// TIA Portal V17 export
// export: Created 2023-04-04T07:17:24.6561318Z, ExportSetting WithDefaults, DisplayName Totally Integrated Automation Portal, DisplayVersion V17 Update 4, DisplayName TIA Portal Openness, DisplayVersion V17 Update 4, DisplayName TIA Portal Version Control Interface, DisplayVersion V17, DisplayName STEP 7 Professional, DisplayVersion V17 Update 4, DisplayName STEP 7 Safety, DisplayVersion V17, DisplayName WinCC Professional, DisplayVersion V17 Update 4
FUNCTION "NTP" : Void   // FC124, LAD
{ S7_Optimized_Access := 'TRUE' }
VERSION : 0.1
// stored: AutoNumber false, IsIECCheckEnabled false, SetENOAutomatically false, UDAEnableTagReadback false
   VAR_TEMP   // added for the SCL form of the ladder/FBD networks
      _w1 : Bool;
   END_VAR
BEGIN

REGION Network 1: Server NTP
   // To run also in a task 1s, it's used by the MINI_PC to retrieve the correct date and time
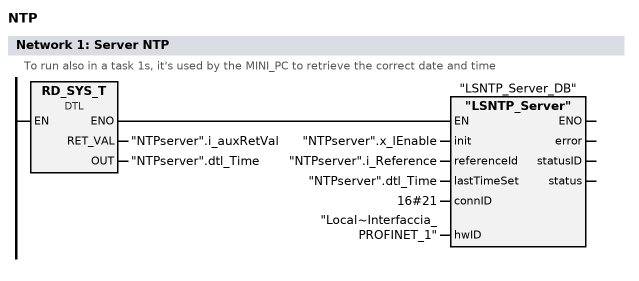
   RUNG wire#powerrail
      { S7_Templates := "date_type := DTL" } RD_SYS_T(RET_VAL => "NTPserver".i_auxRetVal, OUT => "NTPserver".dtl_Time)
      "LSNTP_Server_DB"(init := "NTPserver".x_lEnable, referenceId := "NTPserver".i_Reference, lastTimeSet := "NTPserver".dtl_Time, connID := 16#21, hwID := "Local~Interfaccia_PROFINET_1", error =>, statusID =>, status =>)
   END_RUNG
   // the same network as SCL:
   "NTPserver".i_auxRetVal := RD_SYS_T(OUT => "NTPserver".dtl_Time, ENO => #_w1);
   IF #_w1 THEN
       "LSNTP_Server_DB"(init := "NTPserver".x_lEnable,   // "LSNTP_Server"
                         referenceId := "NTPserver".i_Reference,
                         lastTimeSet := "NTPserver".dtl_Time,
                         connID := 16#21,
                         hwID := "Local~Interfaccia_PROFINET_1");
   END_IF;
END_REGION
END_FUNCTION
